// TIA Portal V20 export
DATA_BLOCK "DB_Motor1"   // DB1
TITLE = DB_Motor1
AUTHOR : Gemini
// stored: InstanceOfName FB_MotorControl, InstanceOfType FB
"FB_MotorControl"
   // VAR_INPUT
   //    bStart : Bool;
   //    bStop : Bool;
   // END_VAR
   // VAR_OUTPUT
   //    bRunning : Bool;
   //    bFault : Bool;
   // END_VAR
   // VAR
   //    tRunTime : Time;
   // END_VAR
BEGIN
END_DATA_BLOCK
